// TIA Portal V20 export
// export: Created 2026-04-11T06:02:30.3209107Z, ExportSetting WithDefaults, DisplayName Totally Integrated Automation Portal, DisplayVersion V20, DisplayName TIA Portal Openness, DisplayVersion V20, DisplayName TIA Portal Version Control Interface, DisplayVersion V20, DisplayName STEP 7 Professional, DisplayVersion V20, DisplayName STEP 7 Safety, DisplayVersion V20, DisplayName WinCC Basic/Comfort/Advanced, DisplayVersion V20, DisplayName WinCC Unified, DisplayVersion V20
TYPE "udtHMI_ValveControl"
// stored: IsFailsafeCompliant false
   STRUCT
      iMode : Int;   // Current mode
      iErrorCode { ExternalWritable := 'False'} : Int;   // Error code
      iStatus { ExternalWritable := 'False'} : Int;   // Status for HMI display
      bPB_ResetError : Bool;   // PB Reset block errors
      bPB_Home : Bool;   // PB Move to home in manual mode
      bPB_Work : Bool;   // PB Move to work in manual mode
      bPBEN_ResetError { ExternalWritable := 'False'} : Bool;   // PB Reset error enabled
      bPBEN_Home { ExternalWritable := 'False'} : Bool;   // PB Home enabled
      bPBEN_Work { ExternalWritable := 'False'} : Bool;   // PB Work enabled
      bHomeOn { ExternalWritable := 'False'} : Bool;   // Home command is on
      bWorkOn { ExternalWritable := 'False'} : Bool;   // Work command is on
      bSignalHome { ExternalWritable := 'False'} : Bool;   // Home feedback
      bSignalWork { ExternalWritable := 'False'} : Bool;   // Work feedback
      bError { ExternalWritable := 'False'} : Bool;   // Error status
      bInterlock { ExternalWritable := 'False'} : Bool;   // Valve interlocked
   END_STRUCT;
END_TYPE
